FUNCTION Convert_LREAL_TO_REAL : Hresult
VAR_INPUT
	in : LREAL;
	out : REFERENCE TO REAL;
END_VAR
VAR
	converted : REAL;
END_VAR

IF (in < -3.402823E+38) THEN	
	Convert_LREAL_TO_REAL := INCOMPATIBLE;
	RETURN;	
END_IF

IF (in > 3.402823E+38) THEN	
	Convert_LREAL_TO_REAL := INCOMPATIBLE;
	RETURN;	
END_IF

out := LREAL_TO_REAL(in);

END_FUNCTION

(* stored: Version 1.1.0.1, ProductVersion 3.1.4024.12
   POU Convert_LREAL_TO_REAL: Id {5a0040ab-68dd-44bb-8f73-70d7d9fb15ac}, SpecialFunc None *)
